{attribute 'linkalways'} 
{attribute 'no_explicit_call' := 'This FB is a CLASS and must be accessed using methods or properties'}
{attribute 'enable_dynamic_creation'}
FUNCTION_BLOCK Node_F_VN_MaxElementElementwise_DINT EXTENDS VisionNode
VAR
    ipContainer : _ITcVnContainer;
    nMax : _DINT(0);
    hrPrev : _HRESULT(S_OK);
    hresult : _HRESULT(S_OK);
END_VAR

METHOD PUBLIC  Clone : I_Node
VAR
	pNode : POINTER TO Node_F_VN_MaxElementElementwise_DINT;
END_VAR
pNode := __NEW(Node_F_VN_MaxElementElementwise_DINT);
Clone := pNode^;
END_METHOD

METHOD FB_init : BOOL
VAR_INPUT
	bInitRetains : BOOL; // if TRUE, the retain variables are initialized (warm start / cold start)
	bInCopyCode : BOOL;  // if TRUE, the instance afterwards gets moved into the copy code (online change)
END_VAR
AddInput('ipContainer', ipContainer);
AddInput('nMax', nMax);
AddInput('hrPrev', hrPrev);
AddOutput('ipContainer', ipContainer);
AddOutput('hresult',hresult);
END_METHOD

METHOD PROTECTED OnExecute : HRESULT
hresult.Value := F_VN_MaxElementElementwise_DINT(
    ipContainer := ipContainer.Value,
    nMax := nMax.Value,
    hrPrev:= hrPrev.Value);
END_METHOD

METHOD PUBLIC PreExecutionCheck
VAR_INPUT
	Check : I_PreExecutionChecks;
END_VAR
Check.IsTrue(ipContainer.IsValid, 'ipContainer must be a valid container');
END_METHOD

END_FUNCTION_BLOCK

(* stored: Version 1.1.0.1, ProductVersion 3.1.4024.13
   POU Node_F_VN_MaxElementElementwise_DINT: Id {21c6779e-c291-43ba-a742-d6ea76d33d91}, SpecialFunc None
   Folder Constructor: Id {f9d07ee2-83d6-4c3b-83ae-5e12f7ca850f}
   Method Clone: Id {c7498aad-08cf-49b4-a9e3-4e75e031261f}
   Method FB_init: Id {c17c35ca-edbb-4120-a200-ed9410924392}
   Method OnExecute: Id {11b8b007-d97c-451f-a913-3d3a93e19cfc}
   Method PreExecutionCheck: Id {f2245620-52c5-4fb9-b523-f60bacb0b035} *)
